FUNCTION_BLOCK FB_Robot
VAR_INPUT
	
	inint_NoOfJobs			: INT; 					(*	Number of Jobs / Numarul de module 	*)
	ins_CommIn				: Type_CommIn_Robot; 	(*	Communication Input for Robot / Modulele de comunicare pentru robot *)
	inint_OptNextJob		:INT;
	inm_Reset				:BOOL;
	
	inCom_0					:BOOL;	
	inCom_1					:BOOL;
	inCom_2					:BOOL;	
	inCom_3					:BOOL;	
	inCom_4					:BOOL;	
	inCom_5					:BOOL;	
	inCom_6					:BOOL;	
	inCom_7					:BOOL;	
	
	inCom_Re_0				:BYTE;
	inCom_Re_1				:BYTE;
	inCom_Re_2				:BYTE;
	inCom_Re_3				:BYTE;
	inCom_Re_4				:BYTE;
	inCom_Re_5				:BYTE;
	inCom_Re_6				:BYTE;
	inCom_Re_7				:BYTE;
	
	in_Opt					:Type_CommIn_Optimization;

END_VAR

VAR_OUTPUT

	outs_Order				: ENUM_OrderState;		(*	State of the order 0-Working / 1-Done / Starea actuala a piesei ridicate 0-in aer / 1-terminata *)
	outs_CommOut			: Type_CommOut_Robot;	(*	Communication output from robot / Comunicarea de la robot catre celelalte module *)
	m_Busy					: BOOL;					(*	Control variable that signals all the modules that robot is busy / o variabila de control ce semnalizeaza tuturor celorlalte module ca robotul este ocupat *)
	outs_Reset				: Type_CommOut_Reset;
	
	outs_Job				:ENUM_Order;
	outint_LastPosition		:INT;
	outdword_StartTime		:Type_Opt_Timers;
	outreal_AverageCycleTime:Type_Opt_CycleTime;
	out_Availabilty			:Type_OptIn_Availability;
	
	outCom_0				:BOOL 	:= m_CallRobotToModule[0];
	outCom_1				:BOOL	:= m_GoDownPick;
	outCom_2				:BOOL	:= m_CallRobotToModule[2];
	outCom_3				:BOOL	:= m_CallRobotToModule[3];
	outCom_4				:BOOL	:= m_CallRobotToModule[4];
	outCom_5				:BOOL	:= m_CallRobotToModule[5];
	outCom_6				:BOOL	:= m_CallRobotToModule[6];
	outCom_7				:BOOL	:= m_GoDownPlace;
	
	
	outCOm_Re_0				:BYTE;
	outCom_Re_1				:BYTE;
	outCom_Re_2				:BYTE;
	outCom_Re_3				:BYTE;
	outCom_Re_4				:BYTE	:=BOOL_TO_BYTE(m_CallRobotToModule[1]);
	outCom_Re_5				:BYTE;
	outCom_Re_6				:BYTE;
	outCom_Re_7				:BYTE;
	
	
END_VAR		

VAR
	Position		: ARRAY [0..11] OF BOOL; (*	Tine minte numarul modulului in dreptul caruia se afla robotul.In acelasi timp, 
											daca un index este egal cu 1, inseamna ca la modulul respectiv se va lucra,
											Se va face Pick sau Place*) 		
	int_Index				: INT;						(*	Index for memorizing the positions*)
	int_IndexForward		: INT;
	int_NextOrder			: ENUM_Order;				(*	*)
	int_PreviousOrder		: ENUM_Order;
	int_LastPosition		: INT;
	int_OptValue			: INT;
	MovementTimes			: ARRAY [0..50] OF TYPE_MovementTime;
	MovementTimesForward	: ARRAY [0..50] OF TYPE_MovementTime;
	m_BaseFinished			: BOOL :=TRUE;
	m_Picked				: BOOL;						(*	Daca robotul a executat miscarea de ridicare a piesei Down->Catch->Up, m_Picked devine true*)
	m_Placed				: BOOL;
	m_GoNextModule			: BOOL;						(*	Variabila de control pentru robot (in val3 citesc valoarea acestei variabile pentru a stii daca incep deplasarea sau nu)*)
	
	m_CallRobotToModule	:ARRAY[0..11] OF BOOL;		(*	Un array de bool prin care chem robotul la modulul la care am nevoie de el *)
	m_Condition			:BOOL;
	
	m_OptOn				:BOOL;
	
	T_Conveyor			:TON;
	T_Test1				:TON;
	T_Test2				:TON;
	T_Test3				:TON;
	T_Drilling1			:TON;
	T_Drilling			:TON;
	
	TC_StartTime		:DWORD;
	T1_StartTime		:DWORD;
	T2_StartTime		:DWORD;
	T3_StartTime		:DWORD;
	TD_StartTime		:DWORD;
	TD1_StartTime		:DWORD;
	
	T01_HelpTimer		:TON;
	T02_MoveTimer		:TON;
	T02_MoveTimer1		:TON;
	
	m_GoDownPick	:BOOL;	(*	Variabila ce transmite robotului ca poate face miscarea de pick*)
	m_GoDownPlace	:BOOL;	(*	Variabila ce transmite robotului ca poate face miscarea de place*)
	
	RetVal				: enum_RetVal;
	
	SFCInit 			:BOOL;
	(*-- Add IN/OUT for Robot Ethercat Communication	*)
	
	(* IN	*)	
	In_0_Byte_0_Bit_0	AT %I* 		:BOOL;
	In_0_Byte_0_Bit_1	AT %I* 		:BOOL;
	In_0_Byte_0_Bit_2	AT %I* 		:BOOL;
	In_0_Byte_0_Bit_3	AT %I* 		:BOOL;
	In_0_Byte_0_Bit_4	AT %I* 		:BOOL;
	In_0_Byte_0_Bit_5	AT %I* 		:BOOL;
	In_0_Byte_0_Bit_6	AT %I* 		:BOOL;
	In_0_Byte_0_Bit_7	AT %I* 		:BOOL;
	
	(* IN REAL*)
	
	inRe_0_Byte_0			AT %I*		:BYTE;
	inRe_0_Byte_1			AT %I*		:BYTE;
	inRe_0_Byte_2			AT %I*		:BYTE;
	inRe_0_Byte_3			AT %I*		:BYTE;
	inRe_0_Byte_4			AT %I*		:BYTE;
	inRe_0_Byte_5			AT %I*		:BYTE;
	inRe_0_Byte_6			AT %I*		:BYTE;
	inRe_0_Byte_7			AT %I*		:BYTE;


	(*	OUT	*)
	Out_0_Byte_0_Bit_0	AT %Q* 		:BOOL;
	Out_0_Byte_0_Bit_1	AT %Q* 		:BOOL;
	Out_0_Byte_0_Bit_2	AT %Q* 		:BOOL;
	Out_0_Byte_0_Bit_3	AT %Q* 		:BOOL;
	Out_0_Byte_0_Bit_4	AT %Q* 		:BOOL;
	Out_0_Byte_0_Bit_5	AT %Q* 		:BOOL;
	Out_0_Byte_0_Bit_6	AT %Q* 		:BOOL;
	Out_0_Byte_0_Bit_7	AT %Q* 		:BOOL;
	
	(* OUT REAL*)
	
	outRe_0_Byte_0			AT %Q*		:BYTE;
	outRe_0_Byte_1			AT %Q*		:BYTE;
	outRe_0_Byte_2			AT %Q*		:BYTE;
	outRe_0_Byte_3			AT %Q*		:BYTE;
	outRe_0_Byte_4			AT %Q*		:BYTE;
	outRe_0_Byte_5			AT %Q*		:BYTE;
	outRe_0_Byte_6			AT %Q*		:BYTE;
	outRe_0_Byte_7			AT %Q*		:BYTE;

	(*--											  --*)
	
	Inst_MovementTime			:FB_RobotMovementTime();
	Inst_MovementTimeBack		:FB_RobotMovementTime();
	
	Inst_Count5PiecesDone		:FB_CountCycleTime();
	real_PiecesTime				:REAL;
	int_PartsDone				:INT;	

END_VAR

A98_SetOutputs();
A99_Communication();

IF NOT inm_Reset 
	THEN
	m_Condition:=FALSE;
	Inst_MovementTime();
	Inst_MovementTimeBack();
	A02_AutomaticMode();
	
ELSIF inm_Reset 
	THEN
	
	IF NOT m_Condition
		THEN
		SFCReset:=TRUE;
		A02_AutomaticMode();		
	END_IF
	
	m_Condition:=TRUE;
	A03_S2_Reset();

END_IF

ACTION A02_AutomaticMode:
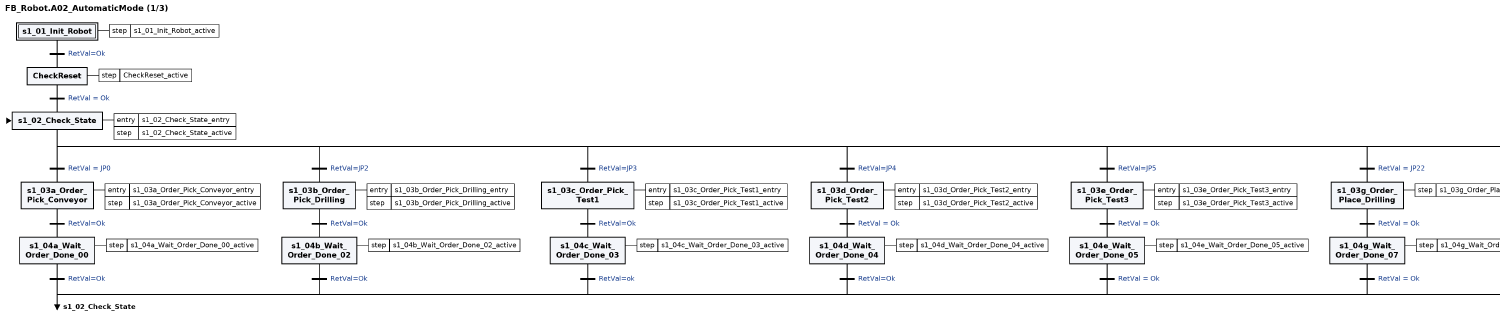
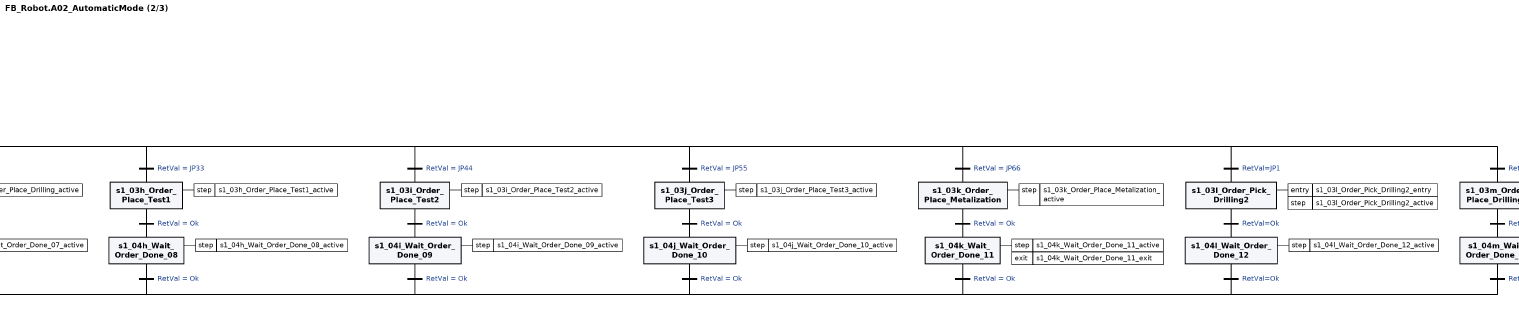
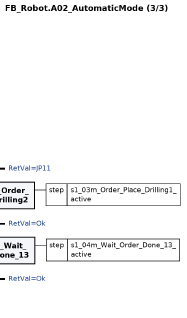
INITIAL_STEP s1_01_Init_Robot:
    s1_01_Init_Robot_active(N);  // step action
END_STEP
TRANSITION FROM s1_01_Init_Robot TO CheckReset
    := RetVal=Ok;
END_TRANSITION
STEP CheckReset:
    CheckReset_active(N);  // step action
END_STEP
TRANSITION FROM CheckReset TO s1_02_Check_State
    := RetVal = Ok;
END_TRANSITION
STEP s1_02_Check_State:
    s1_02_Check_State_entry(P1);  // entry action
    s1_02_Check_State_active(N);  // step action
END_STEP
TRANSITION FROM s1_02_Check_State TO s1_03a_Order_Pick_Conveyor
    := RetVal = JP0;
END_TRANSITION
STEP s1_03a_Order_Pick_Conveyor:
    s1_03a_Order_Pick_Conveyor_entry(P1);  // entry action
    s1_03a_Order_Pick_Conveyor_active(N);  // step action
END_STEP
TRANSITION FROM s1_03a_Order_Pick_Conveyor TO s1_04a_Wait_Order_Done_00
    := RetVal=Ok;
END_TRANSITION
STEP s1_04a_Wait_Order_Done_00:
    s1_04a_Wait_Order_Done_00_active(N);  // step action
END_STEP
TRANSITION FROM s1_04a_Wait_Order_Done_00 TO s1_02_Check_State
    := RetVal=Ok;
END_TRANSITION
TRANSITION FROM s1_02_Check_State TO s1_03b_Order_Pick_Drilling
    := RetVal=JP2;
END_TRANSITION
STEP s1_03b_Order_Pick_Drilling:
    s1_03b_Order_Pick_Drilling_entry(P1);  // entry action
    s1_03b_Order_Pick_Drilling_active(N);  // step action
END_STEP
TRANSITION FROM s1_03b_Order_Pick_Drilling TO s1_04b_Wait_Order_Done_02
    := RetVal=Ok;
END_TRANSITION
STEP s1_04b_Wait_Order_Done_02:
    s1_04b_Wait_Order_Done_02_active(N);  // step action
END_STEP
TRANSITION FROM s1_04b_Wait_Order_Done_02 TO s1_02_Check_State
    := RetVal=Ok;
END_TRANSITION
TRANSITION FROM s1_02_Check_State TO s1_03c_Order_Pick_Test1
    := RetVal=JP3;
END_TRANSITION
STEP s1_03c_Order_Pick_Test1:
    s1_03c_Order_Pick_Test1_entry(P1);  // entry action
    s1_03c_Order_Pick_Test1_active(N);  // step action
END_STEP
TRANSITION FROM s1_03c_Order_Pick_Test1 TO s1_04c_Wait_Order_Done_03
    := RetVal=Ok;
END_TRANSITION
STEP s1_04c_Wait_Order_Done_03:
    s1_04c_Wait_Order_Done_03_active(N);  // step action
END_STEP
TRANSITION FROM s1_04c_Wait_Order_Done_03 TO s1_02_Check_State
    := RetVal=ok;
END_TRANSITION
TRANSITION FROM s1_02_Check_State TO s1_03d_Order_Pick_Test2
    := RetVal=JP4;
END_TRANSITION
STEP s1_03d_Order_Pick_Test2:
    s1_03d_Order_Pick_Test2_entry(P1);  // entry action
    s1_03d_Order_Pick_Test2_active(N);  // step action
END_STEP
TRANSITION FROM s1_03d_Order_Pick_Test2 TO s1_04d_Wait_Order_Done_04
    := RetVal = Ok;
END_TRANSITION
STEP s1_04d_Wait_Order_Done_04:
    s1_04d_Wait_Order_Done_04_active(N);  // step action
END_STEP
TRANSITION FROM s1_04d_Wait_Order_Done_04 TO s1_02_Check_State
    := RetVal=Ok;
END_TRANSITION
TRANSITION FROM s1_02_Check_State TO s1_03e_Order_Pick_Test3
    := RetVal=JP5;
END_TRANSITION
STEP s1_03e_Order_Pick_Test3:
    s1_03e_Order_Pick_Test3_entry(P1);  // entry action
    s1_03e_Order_Pick_Test3_active(N);  // step action
END_STEP
TRANSITION FROM s1_03e_Order_Pick_Test3 TO s1_04e_Wait_Order_Done_05
    := RetVal = Ok;
END_TRANSITION
STEP s1_04e_Wait_Order_Done_05:
    s1_04e_Wait_Order_Done_05_active(N);  // step action
END_STEP
TRANSITION FROM s1_04e_Wait_Order_Done_05 TO s1_02_Check_State
    := RetVal = Ok;
END_TRANSITION
TRANSITION FROM s1_02_Check_State TO s1_03g_Order_Place_Drilling
    := RetVal = JP22;
END_TRANSITION
STEP s1_03g_Order_Place_Drilling:
    s1_03g_Order_Place_Drilling_active(N);  // step action
END_STEP
TRANSITION FROM s1_03g_Order_Place_Drilling TO s1_04g_Wait_Order_Done_07
    := RetVal = Ok;
END_TRANSITION
STEP s1_04g_Wait_Order_Done_07:
    s1_04g_Wait_Order_Done_07_active(N);  // step action
END_STEP
TRANSITION FROM s1_04g_Wait_Order_Done_07 TO s1_02_Check_State
    := RetVal = Ok;
END_TRANSITION
TRANSITION FROM s1_02_Check_State TO s1_03h_Order_Place_Test1
    := RetVal = JP33;
END_TRANSITION
STEP s1_03h_Order_Place_Test1:
    s1_03h_Order_Place_Test1_active(N);  // step action
END_STEP
TRANSITION FROM s1_03h_Order_Place_Test1 TO s1_04h_Wait_Order_Done_08
    := RetVal = Ok;
END_TRANSITION
STEP s1_04h_Wait_Order_Done_08:
    s1_04h_Wait_Order_Done_08_active(N);  // step action
END_STEP
TRANSITION FROM s1_04h_Wait_Order_Done_08 TO s1_02_Check_State
    := RetVal = Ok;
END_TRANSITION
TRANSITION FROM s1_02_Check_State TO s1_03i_Order_Place_Test2
    := RetVal = JP44;
END_TRANSITION
STEP s1_03i_Order_Place_Test2:
    s1_03i_Order_Place_Test2_active(N);  // step action
END_STEP
TRANSITION FROM s1_03i_Order_Place_Test2 TO s1_04i_Wait_Order_Done_09
    := RetVal = Ok;
END_TRANSITION
STEP s1_04i_Wait_Order_Done_09:
    s1_04i_Wait_Order_Done_09_active(N);  // step action
END_STEP
TRANSITION FROM s1_04i_Wait_Order_Done_09 TO s1_02_Check_State
    := RetVal = Ok;
END_TRANSITION
TRANSITION FROM s1_02_Check_State TO s1_03j_Order_Place_Test3
    := RetVal = JP55;
END_TRANSITION
STEP s1_03j_Order_Place_Test3:
    s1_03j_Order_Place_Test3_active(N);  // step action
END_STEP
TRANSITION FROM s1_03j_Order_Place_Test3 TO s1_04j_Wait_Order_Done_10
    := RetVal = Ok;
END_TRANSITION
STEP s1_04j_Wait_Order_Done_10:
    s1_04j_Wait_Order_Done_10_active(N);  // step action
END_STEP
TRANSITION FROM s1_04j_Wait_Order_Done_10 TO s1_02_Check_State
    := RetVal = Ok;
END_TRANSITION
TRANSITION FROM s1_02_Check_State TO s1_03k_Order_Place_Metalization
    := RetVal = JP66;
END_TRANSITION
STEP s1_03k_Order_Place_Metalization:
    s1_03k_Order_Place_Metalization_active(N);  // step action
END_STEP
TRANSITION FROM s1_03k_Order_Place_Metalization TO s1_04k_Wait_Order_Done_11
    := RetVal = Ok;
END_TRANSITION
STEP s1_04k_Wait_Order_Done_11:
    s1_04k_Wait_Order_Done_11_active(N);  // step action
    s1_04k_Wait_Order_Done_11_exit(P0);  // exit action
END_STEP
TRANSITION FROM s1_04k_Wait_Order_Done_11 TO s1_02_Check_State
    := RetVal = Ok;
END_TRANSITION
TRANSITION FROM s1_02_Check_State TO s1_03l_Order_Pick_Drilling2
    := RetVal=JP1;
END_TRANSITION
STEP s1_03l_Order_Pick_Drilling2:
    s1_03l_Order_Pick_Drilling2_entry(P1);  // entry action
    s1_03l_Order_Pick_Drilling2_active(N);  // step action
END_STEP
TRANSITION FROM s1_03l_Order_Pick_Drilling2 TO s1_04l_Wait_Order_Done_12
    := RetVal=Ok;
END_TRANSITION
STEP s1_04l_Wait_Order_Done_12:
    s1_04l_Wait_Order_Done_12_active(N);  // step action
END_STEP
TRANSITION FROM s1_04l_Wait_Order_Done_12 TO s1_02_Check_State
    := RetVal=Ok;
END_TRANSITION
TRANSITION FROM s1_02_Check_State TO s1_03m_Order_Place_Drilling2
    := RetVal=JP11;
END_TRANSITION
STEP s1_03m_Order_Place_Drilling2:
    s1_03m_Order_Place_Drilling1_active(N);  // step action
END_STEP
TRANSITION FROM s1_03m_Order_Place_Drilling2 TO s1_04m_Wait_Order_Done_13
    := RetVal=Ok;
END_TRANSITION
STEP s1_04m_Wait_Order_Done_13:
    s1_04m_Wait_Order_Done_13_active(N);  // step action
END_STEP
TRANSITION FROM s1_04m_Wait_Order_Done_13 TO s1_02_Check_State
    := RetVal=Ok;
END_TRANSITION
// branch label Branch0_A01_AutomaticMode
END_ACTION

ACTION A03_S2_Reset:
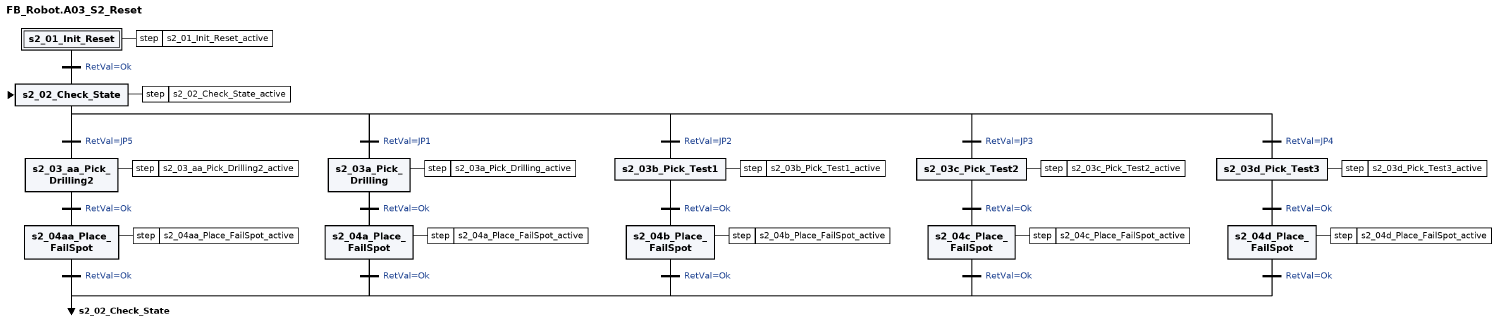
INITIAL_STEP s2_01_Init_Reset:
    s2_01_Init_Reset_active(N);  // step action
END_STEP
TRANSITION FROM s2_01_Init_Reset TO s2_02_Check_State
    := RetVal=Ok;
END_TRANSITION
STEP s2_02_Check_State:
    s2_02_Check_State_active(N);  // step action
END_STEP
TRANSITION FROM s2_02_Check_State TO s2_03_aa_Pick_Drilling2
    := RetVal=JP5;
END_TRANSITION
STEP s2_03_aa_Pick_Drilling2:
    s2_03_aa_Pick_Drilling2_active(N);  // step action
END_STEP
TRANSITION FROM s2_03_aa_Pick_Drilling2 TO s2_04aa_Place_FailSpot
    := RetVal=Ok;
END_TRANSITION
STEP s2_04aa_Place_FailSpot:
    s2_04aa_Place_FailSpot_active(N);  // step action
END_STEP
TRANSITION FROM s2_04aa_Place_FailSpot TO s2_02_Check_State
    := RetVal=Ok;
END_TRANSITION
TRANSITION FROM s2_02_Check_State TO s2_03a_Pick_Drilling
    := RetVal=JP1;
END_TRANSITION
STEP s2_03a_Pick_Drilling:
    s2_03a_Pick_Drilling_active(N);  // step action
END_STEP
TRANSITION FROM s2_03a_Pick_Drilling TO s2_04a_Place_FailSpot
    := RetVal=Ok;
END_TRANSITION
STEP s2_04a_Place_FailSpot:
    s2_04a_Place_FailSpot_active(N);  // step action
END_STEP
TRANSITION FROM s2_04a_Place_FailSpot TO s2_02_Check_State
    := RetVal=Ok;
END_TRANSITION
TRANSITION FROM s2_02_Check_State TO s2_03b_Pick_Test1
    := RetVal=JP2;
END_TRANSITION
STEP s2_03b_Pick_Test1:
    s2_03b_Pick_Test1_active(N);  // step action
END_STEP
TRANSITION FROM s2_03b_Pick_Test1 TO s2_04b_Place_FailSpot
    := RetVal=Ok;
END_TRANSITION
STEP s2_04b_Place_FailSpot:
    s2_04b_Place_FailSpot_active(N);  // step action
END_STEP
TRANSITION FROM s2_04b_Place_FailSpot TO s2_02_Check_State
    := RetVal=Ok;
END_TRANSITION
TRANSITION FROM s2_02_Check_State TO s2_03c_Pick_Test2
    := RetVal=JP3;
END_TRANSITION
STEP s2_03c_Pick_Test2:
    s2_03c_Pick_Test2_active(N);  // step action
END_STEP
TRANSITION FROM s2_03c_Pick_Test2 TO s2_04c_Place_FailSpot
    := RetVal=Ok;
END_TRANSITION
STEP s2_04c_Place_FailSpot:
    s2_04c_Place_FailSpot_active(N);  // step action
END_STEP
TRANSITION FROM s2_04c_Place_FailSpot TO s2_02_Check_State
    := RetVal=Ok;
END_TRANSITION
TRANSITION FROM s2_02_Check_State TO s2_03d_Pick_Test3
    := RetVal=JP4;
END_TRANSITION
STEP s2_03d_Pick_Test3:
    s2_03d_Pick_Test3_active(N);  // step action
END_STEP
TRANSITION FROM s2_03d_Pick_Test3 TO s2_04d_Place_FailSpot
    := RetVal=Ok;
END_TRANSITION
STEP s2_04d_Place_FailSpot:
    s2_04d_Place_FailSpot_active(N);  // step action
END_STEP
TRANSITION FROM s2_04d_Place_FailSpot TO s2_02_Check_State
    := RetVal=Ok;
END_TRANSITION
// branch label Branch0_A03_S2_Reset
END_ACTION

ACTION A98_SetOutputs:
outCom_0	:= inCom_0;
outCom_1 	:= inCom_1;
outCom_2 	:= inCom_2;
outCom_3 	:= inCom_3;
outCom_4 	:= inCom_4;
outCom_5	:= inCom_5;
outCom_6 	:= inCom_6;
outCom_7 	:= inCom_7;


outCom_Re_0	:= inCom_Re_0;
outCom_Re_1	:= inCom_Re_1;
outCom_Re_2	:= inCom_Re_2;
outCom_Re_3	:= inCom_Re_3;
outCom_Re_4	:= inCom_Re_4;
outCom_Re_5	:= inCom_Re_5;
outCom_Re_6	:= inCom_Re_6;
outCom_Re_7	:= inCom_Re_7;
END_ACTION

ACTION A99_Communication:

(*inputs*)

Position[0] 	:= In_0_Byte_0_Bit_0;
m_Picked 		:= In_0_Byte_0_Bit_1;
Position[2]  	:= In_0_Byte_0_Bit_2;
Position[3]  	:= In_0_Byte_0_Bit_3;
Position[4]  	:= In_0_Byte_0_Bit_4;
Position[5]  	:= In_0_Byte_0_Bit_5;
Position[6]  	:= In_0_Byte_0_Bit_6;
m_Placed 		:= In_0_Byte_0_Bit_7;


inCom_Re_0		:= inRe_0_Byte_0;
inCom_Re_1		:= inRe_0_Byte_1;
inCom_Re_2		:= inRe_0_Byte_2;
inCom_Re_3		:= inRe_0_Byte_3;
Position[1]		:= BYTE_TO_BOOL(inRe_0_Byte_4);
m_OptOn			:= BYTE_TO_BOOL(inRe_0_Byte_5);
inCom_Re_6		:= inRe_0_Byte_6;
inCom_Re_7		:= inRe_0_Byte_7;

(*outputs*)

Out_0_Byte_0_Bit_0 	:= m_CallRobotToModule[0];
Out_0_Byte_0_Bit_1 	:= m_GoDownPick;
Out_0_Byte_0_Bit_2 	:= m_CallRobotToModule[2];
Out_0_Byte_0_Bit_3 	:= m_CallRobotToModule[3];
Out_0_Byte_0_Bit_4	:= m_CallRobotToModule[4];
Out_0_Byte_0_Bit_5 	:= m_CallRobotToModule[5];
Out_0_Byte_0_Bit_6 	:= m_CallRobotToModule[6];
Out_0_Byte_0_Bit_7 	:= m_GoDownPlace;

outRe_0_Byte_0		:= outCom_Re_0;
outRe_0_Byte_1		:= outCom_Re_1;
outRe_0_Byte_2		:= outCom_Re_2;
outRe_0_Byte_3		:= outCom_Re_3;
outRe_0_Byte_4		:= BOOL_TO_BYTE(m_CallRobotToModule[1]);
outRe_0_Byte_5		:= INT_TO_BYTE(int_OptValue);
outRe_0_Byte_6		:= outCom_Re_6;
outRe_0_Byte_7		:= outCom_Re_7;

outdword_StartTime.T_Conveyor	:=TC_StartTime;
outdword_StartTime.T_Drilling_1	:=TD1_StartTime;
outdword_StartTime.T_Drilling	:=TD_StartTime;
outdword_StartTime.T_Test_1		:=T1_StartTime;
outdword_StartTime.T_Test_2		:=T2_StartTime;
outdword_StartTime.T_Test_3		:=T3_StartTime;

outreal_AverageCycleTime.re_Conveyor	:=in_Opt.s_Conveyor.out_AverageCycleTime;
outreal_AverageCycleTime.re_Drilling_1	:=in_Opt.s_Drilling_1.out_AverageCycleTime;
outreal_AverageCycleTime.re_Drilling	:=in_Opt.s_Drilling_2.out_AverageCycleTime;
outreal_AverageCycleTime.re_Test_1		:=in_Opt.s_Test_1.out_AverageCycleTime;
outreal_AverageCycleTime.re_Test_2		:=in_Opt.s_Test_2.out_AverageCycleTime;
outreal_AverageCycleTime.re_Test_3		:=in_Opt.s_Test_3.out_AverageCycleTime;

out_Availabilty.s_Drilling_1.m_Available	:= ins_CommIn.s_Drilling.m_Empty;
out_Availabilty.s_Drilling_2.m_Available	:= ins_CommIn.s_Drilling1.m_Empty;
out_Availabilty.s_Test_1.m_Available		:= ins_CommIn.s_Test_1.m_Empty;
out_Availabilty.s_Test_2.m_Available		:= ins_CommIn.s_Test_2.m_Empty;
out_Availabilty.s_Test_3.m_Available		:= ins_CommIn.s_Test_3.m_Empty;
out_Availabilty.s_Metalization.m_Available	:= ins_CommIn.s_Metalization.m_Empty;

outint_LastPosition	:=int_LastPosition;
outs_Job			:=int_NextOrder;
END_ACTION

ACTION CheckReset_active:
RetVal	:=Running;

IF 	NOT inm_Reset
	THEN
	RetVal	:=Ok;
END_IF
END_ACTION

ACTION s1_01_Init_Robot_active:
IF m_BaseFinished
	THEN	
		Inst_Count5PiecesDone(inm_TimeActive:=TRUE);
		
		outs_Order:=ENUM_OrderState.Done;
		
		outs_CommOut.s_Conveyor.m_OutOfArea		:=TRUE;
		outs_CommOut.s_Drilling.m_OutOfArea		:=TRUE;	
		outs_CommOut.s_Drilling1.m_OutOfArea	:=TRUE;	
		outs_CommOut.s_Test_1.m_OutOfArea		:=TRUE;
		outs_CommOut.s_Test_2.m_OutOfArea		:=TRUE;
		outs_CommOut.s_Test_3.m_OutOfArea		:=TRUE;
		outs_CommOut.s_Metalization.m_OutOfArea	:=TRUE;
		
		outs_Reset.outm_Reset_Drilling	:=FALSE;
		outs_Reset.outm_Reset_Drilling2	:=FALSE;
		outs_Reset.outm_Reset_Test1		:=FALSE;
		outs_Reset.outm_Reset_Test2		:=FALSE;
		outs_Reset.outm_Reset_Test3		:=FALSE;

		T1_StartTime:=T2_StartTime:=T3_StartTime:=	TIME_TO_DWORD(T#1D) + 20000;
		TD1_StartTime:=TD_StartTime:=TC_StartTime:= TIME_TO_DWORD(T#1D);
		
		RetVal:=Ok;
		
		
			
END_IF
END_ACTION

ACTION s1_02_Check_State_active:

(* 	----PICK TEST1,TEST2,TEST3----	*)

	IF (	T1_StartTime<T2_StartTime
		AND 	T1_StartTime<T3_StartTime)
		AND 	ins_CommIn.s_Test_1.m_Ready
		AND 	ins_CommIn.s_Metalization.m_Empty
		AND NOT m_Picked
		AND (
				int_NextOrder = ENUM_Order.NoOrder
		OR		int_NextOrder = ENUM_Order.Pick_Test_1)
		THEN
			int_NextOrder:=ENUM_Order.Pick_Test_1;
			RetVal := JP3;	
			
	
	ELSIF 	(	T2_StartTime<T1_StartTime
		AND 	T2_StartTime<T3_StartTime)
		AND 	ins_CommIn.s_Test_2.m_Ready
		AND 	ins_CommIn.s_Metalization.m_Empty
		AND NOT m_Picked
		AND (
				int_NextOrder = ENUM_Order.NoOrder
		OR		int_NextOrder = ENUM_Order.Pick_Test_2)
		THEN
			int_NextOrder:=ENUM_Order.Pick_Test_2;
			RetVal := JP4;	
			
	ELSIF 	(	T3_StartTime<T1_StartTime
		AND 	T3_StartTime<T2_StartTime)
		AND 	ins_CommIn.s_Test_3.m_Ready
		AND 	ins_CommIn.s_Metalization.m_Empty	
		AND NOT m_Picked
		AND (
				int_NextOrder = ENUM_Order.NoOrder
		OR		int_NextOrder = ENUM_Order.Pick_Test_3)
		THEN
			int_NextOrder:=ENUM_Order.Pick_Test_3;
			RetVal := JP5;	
	
	
			
	(* 	----PICK DRILLING1,DRILLING2----	*)	
	ELSIF 	TD_StartTime<TD1_StartTime
		AND (	ins_CommIn.s_Drilling.m_Ready
		AND (	ins_CommIn.s_Test_1.m_Empty
			OR 	ins_CommIn.s_Test_2.m_Empty
			OR 	ins_CommIn.s_Test_3.m_Empty
			)
		AND NOT m_Picked
		AND
			( 	int_NextOrder = ENUM_Order.NoOrder 
		OR		int_NextOrder = ENUM_Order.Pick_Drilling)
			)
		THEN
			int_NextOrder:=ENUM_Order.Pick_Drilling;
			RetVal := JP2;
				
	ELSIF 		TD1_StartTime<TD_StartTime
		AND (	ins_CommIn.s_Drilling1.m_Ready
		AND (	ins_CommIn.s_Test_1.m_Empty
			OR 	ins_CommIn.s_Test_2.m_Empty
			OR 	ins_CommIn.s_Test_3.m_Empty
			)
		AND NOT m_Picked
		AND
			( 	int_NextOrder = ENUM_Order.NoOrder 
		OR		int_NextOrder = ENUM_Order.Pick_Drilling1)
			)
		THEN
			int_NextOrder:=ENUM_Order.Pick_Drilling1;
			RetVal := JP1;
			
	(* 	----PICK CONVEYOR----	*)			
	ELSIF		(ins_CommIn.s_Conveyor.m_Ready (* verific daca modulul actual are piesa gata	*)
		AND 	(ins_CommIn.s_Drilling.m_Empty (* verific daca urmatorul modul e gol	(altfel nu fac pick de aici)	*)
		OR		 ins_CommIn.s_Drilling1.m_Empty)
		AND NOT m_Picked	
		AND
			(	int_NextOrder=ENUM_Order.NoOrder 
		OR 		int_NextOrder=ENUM_Order.Pick_Conveyor)
			)
		THEN
			int_NextOrder:=ENUM_Order.Pick_Conveyor;
			RetVal:=JP0;
				
	(*	PLACE	*)
	
	ELSIF 	ins_CommIn.s_Drilling1.m_Empty
		AND m_Picked	
		AND outs_Order = ENUM_OrderState.Done
		AND m_GoNextModule
		AND
		(	int_NextOrder = ENUM_Order.NoOrder 	
		OR	int_NextOrder = ENUM_Order.Place_Drilling2)	
		
		THEN
			RetVal := JP11;
			
	ELSIF 	ins_CommIn.s_Drilling.m_Empty
		AND m_Picked	
		AND outs_Order = ENUM_OrderState.Done
		AND m_GoNextModule
		AND
		(	int_NextOrder = ENUM_Order.NoOrder 	
		OR	int_NextOrder = ENUM_Order.Place_Drilling)	
		
		THEN
			RetVal := JP22;
	
	ELSIF 	ins_CommIn.s_Test_1.m_Empty
		AND m_Picked
		AND NOT m_Busy	
		AND outs_Order = ENUM_OrderState.Done
		AND m_GoNextModule
		AND
		(	int_NextOrder = ENUM_Order.NoOrder 	
		OR	int_NextOrder = ENUM_Order.Place_Test_1)	
		
		THEN
			RetVal := JP33;
		
	ELSIF 	ins_CommIn.s_Test_2.m_Empty
		AND m_Picked
		AND NOT m_Busy	
		AND outs_Order = ENUM_OrderState.Done
		AND m_GoNextModule
		AND
		(	int_NextOrder = ENUM_Order.NoOrder 	
		OR	int_NextOrder = ENUM_Order.Place_Test_2)	
		
		THEN
			RetVal := JP44;
			
	ELSIF 	ins_CommIn.s_Test_3.m_Empty
		AND m_Picked
		AND NOT m_Busy	
		AND outs_Order = ENUM_OrderState.Done
		AND m_GoNextModule
		AND
		(	int_NextOrder = ENUM_Order.NoOrder 	
		OR	int_NextOrder = ENUM_Order.Place_Test_3)	
		
		THEN
			RetVal := JP55;
			
		
	ELSIF 	ins_CommIn.s_Metalization.m_Empty 
		AND m_Picked
		AND outs_Order = ENUM_OrderState.Done
		AND m_GoNextModule
		AND 
		(	int_NextOrder = ENUM_Order.NoOrder
		OR	int_NextOrder = ENUM_Order.Place_Metalization)
		
		THEN
			RetVal := JP66;
	
	END_IF
END_ACTION

ACTION s1_02_Check_State_entry:
RetVal:= Running;

IF m_OptOn AND int_NextOrder=ENUM_Order.NoOrder
	THEN
	int_OptValue:= inint_OptNextJob;
	
	CASE int_OptValue OF
		0:	int_NextOrder := ENUM_Order.Pick_Conveyor;
		1:	int_NextOrder := ENUM_Order.Pick_Drilling1;
		2:	int_NextOrder := ENUM_Order.Pick_Drilling;
		3:	int_NextOrder := ENUM_Order.Pick_Test_1;
		4:	int_NextOrder := ENUM_Order.Pick_Test_2;
		5:	int_NextOrder := ENUM_Order.Pick_Test_3;
	END_CASE
	
END_IF
			
IF int_NextOrder=ENUM_Order.Pick_Conveyor
		AND ins_CommIn.s_Conveyor.m_Ready 
		THEN
			RetVal:=JP0;
			
	ELSIF int_NextOrder=ENUM_Order.Pick_Drilling
		AND ins_CommIn.s_Drilling.m_Ready 
		THEN
			RetVal:=JP2;
			
	ELSIF int_NextOrder=ENUM_Order.Pick_Drilling1
		AND ins_CommIn.s_Drilling1.m_Ready 
		THEN
			RetVal:=JP1;
			
	ELSIF int_NextOrder=ENUM_Order.Pick_Test_1
		AND ins_CommIn.s_Test_1.m_Ready 
		THEN
			RetVal:=JP3;
	ELSIF int_NextOrder=ENUM_Order.Pick_Test_2
		AND ins_CommIn.s_Test_2.m_Ready 
		THEN
			RetVal:=JP4;
	ELSIF int_NextOrder=ENUM_Order.Pick_Test_3
		AND ins_CommIn.s_Test_3.m_Ready 
		THEN
			RetVal:=JP5;
	END_IF
END_ACTION

ACTION s1_03a_Order_Pick_Conveyor_active:
RetVal:=Running;
outs_CommOut.s_Metalization.m_OutOfArea:=TRUE;
(* semnal pentru urmatorul modul ca robotul lucreaza *)
m_CallRobotToModule[0] := TRUE; (*	Chem robotul la conveyor.Aceasta variabila trebuie sa o citesc in programul robotului*)

outs_Order:=ENUM_OrderState.Working; 
outs_CommOut.s_Conveyor.m_Work:=TRUE;(*	Semnalez conveyorul ca robotul urmeaza sa lucreze in jurul lui	*)
T_Conveyor(IN:=FALSE);
IF Position[0] = 1
	THEN
		Inst_MovementTimeBack(inm_Couting:=FALSE, inint_SecondStation:=0);
		MovementTimes[int_Index].FirstStation := Inst_MovementTimeBack.outs_MovementTime.FirstStation;
		MovementTimes[int_Index].SecondStation := Inst_MovementTimeBack.outs_MovementTime.SecondStation;
		MovementTimes[int_Index].MovementTime := Inst_MovementTimeBack.outs_MovementTime.MovementTime;
		outs_CommOut.s_Conveyor.m_OutOfArea:=FALSE;	
		// Trebuie o variabila care sa dea startul miscarii de pick sau de place. m_GoDown
				(*	In acest punct, robotul a luat piesa si este sus ,m_Picked este conctrolat din staubli*)		
END_IF

IF ins_CommIn.s_Conveyor.m_Ready
		THEN		
	m_GoDownPick:=TRUE;	
	IF m_Picked
	THEN
		m_CallRobotToModule[0]	:=	FALSE;
		outs_CommOut.s_Conveyor.m_Work:=FALSE;	
		m_GoDownPick:= FALSE; 	//aici se face FALSE pentru a nu ramane mereu activa.
		TC_StartTime:=TIME_TO_DWORD(T_Conveyor.StartTime);
		int_Index:=int_Index + 1;		
		RetVal :=Ok;						
		END_IF
END_IF
 (*-----------IAR M_PICKED SE VA FACE TRUE IN STAUBLI---------------------------------------*)

// La final... Next order trebuie sa fie de place pe urmatorul modul int_NextOrder:=ENUM_Order.Place_Drilling;




(*	Miscarea	


	Order = Pick	=> 	Move From Initial Position To Asked Position 	--Gloval_Vars.Order[] 
						Move Down To Take Part							--m_MoveDown 
						Move Up With Part								--m_MoveUp	=>m_Picked
					
	Order = Place	=>	Move From Last Position To Asked Position		-Global_Vars.Order[]
						Move Down To Leave Part							--m_MoveDown
						Move Up Empty									--m_MoveUp	=>m_Placed	
						
	
	SAU
	
	
	Order = Pick 	=> Logica facuta in Staubli include MoveToTarget, MoveDown, MoveUp
	*)
END_ACTION

ACTION s1_03a_Order_Pick_Conveyor_entry:
Inst_MovementTimeBack(inm_Couting:=TRUE, inint_FirstStation:=int_LastPosition);
T_Conveyor(IN:=TRUE);
END_ACTION

ACTION s1_03b_Order_Pick_Drilling_active:
RetVal:=Running;
outs_CommOut.s_Metalization.m_OutOfArea:=TRUE;
int_PreviousOrder:= ENUM_Order.Pick_Drilling;
m_CallRobotToModule[2] := TRUE; 
outs_Order:=ENUM_OrderState.Working; 
outs_CommOut.s_Drilling.m_Work:=TRUE;

IF Position[2] = 1
	THEN	
		Inst_MovementTimeBack(inm_Couting:=FALSE, inint_SecondStation:=2);
		MovementTimes[int_Index].FirstStation := Inst_MovementTimeBack.outs_MovementTime.FirstStation;
		MovementTimes[int_Index].SecondStation := Inst_MovementTimeBack.outs_MovementTime.SecondStation;
		MovementTimes[int_Index].MovementTime := Inst_MovementTimeBack.outs_MovementTime.MovementTime;
		outs_CommOut.s_Drilling.m_OutOfArea:=FALSE;
				
		m_GoDownPick	:=TRUE;		
END_IF

		
IF m_Picked (*	m_Picked este controlata din staubli	*)
		THEN
			m_CallRobotToModule[2]	:=	FALSE;
			outs_CommOut.s_Drilling.m_PartDropped:=FALSE;
			outs_CommOut.s_Drilling.m_Work:=FALSE;
			m_GoDownPick:=FALSE;		
			int_Index:=int_Index + 1;	
			RetVal := Ok;
END_IF
END_ACTION

ACTION s1_03b_Order_Pick_Drilling_entry:
Inst_MovementTimeBack(inm_Couting:=TRUE, inint_FirstStation:=int_LastPosition);
END_ACTION

ACTION s1_03c_Order_Pick_Test1_active:
RetVal:=Running;
outs_CommOut.s_Metalization.m_OutOfArea:=TRUE;
int_PreviousOrder := ENUM_Order.Pick_Test_1;
m_CallRobotToModule[3] := TRUE; 
outs_Order:=ENUM_OrderState.Working; (* inseamna ca piesa e in aer *)
outs_CommOut.s_Test_1.m_Work:=TRUE;
 
IF Position[3] = 1
	THEN
		Inst_MovementTimeBack(inm_Couting:=FALSE, inint_SecondStation:=3);
		MovementTimes[int_Index].FirstStation := Inst_MovementTimeBack.outs_MovementTime.FirstStation;
		MovementTimes[int_Index].SecondStation := Inst_MovementTimeBack.outs_MovementTime.SecondStation;
		MovementTimes[int_Index].MovementTime := Inst_MovementTimeBack.outs_MovementTime.MovementTime;
		outs_CommOut.s_Test_1.m_OutOfArea:=FALSE;
	m_GoDownPick	:=TRUE;	
END_IF
	
			
IF m_Picked (*	m_Picked este controlata din staubli	*)
		THEN
			m_CallRobotToModule[3]	:=	FALSE;
			outs_CommOut.s_Test_1.m_PartDropped:=FALSE;
			outs_CommOut.s_Test_1.m_Work:=FALSE;
			m_GoDownPick:=FALSE;
			int_Index:=int_Index + 1;			
			RetVal := Ok;
END_IF

 
// La final... Next order trebuie sa fie de place pe urmatorul modul int_NextOrder:=ENUM_Order.Place_Drilling;




(*	Miscarea	


	Order = Pick	=> 	Move From Initial Position To Asked Position 	--Gloval_Vars.Order[] 
						Move Down To Take Part							--m_MoveDown 
						Move Up With Part								--m_MoveUp	=>m_Picked
					
	Order = Place	=>	Move From Last Position To Asked Position		-Global_Vars.Order[]
						Move Down To Leave Part							--m_MoveDown
						Move Up Empty									--m_MoveUp	=>m_Placed	
						
	
	SAU
	
	
	Order = Pick 	=> Logica facuta in Staubli include MoveToTarget, MoveDown, MoveUp
	*)
END_ACTION

ACTION s1_03c_Order_Pick_Test1_entry:
Inst_MovementTimeBack(inm_Couting:=TRUE, inint_FirstStation:=int_LastPosition);
END_ACTION

ACTION s1_03d_Order_Pick_Test2_active:
RetVal:=Running;
outs_CommOut.s_Metalization.m_OutOfArea:=TRUE;
(* semnal pentru urmatorul modul ca robotul lucreaza *)
int_PreviousOrder := ENUM_Order.Pick_Test_2;
m_CallRobotToModule[4] := TRUE; 
outs_Order:=ENUM_OrderState.Working; (* inseamna ca piesa e in aer *)
outs_CommOut.s_Test_2.m_Work:=TRUE;

IF Position[4] = 1
	THEN
		Inst_MovementTimeBack(inm_Couting:=FALSE, inint_SecondStation:=4);
		MovementTimes[int_Index].FirstStation := Inst_MovementTimeBack.outs_MovementTime.FirstStation;
		MovementTimes[int_Index].SecondStation := Inst_MovementTimeBack.outs_MovementTime.SecondStation;
		MovementTimes[int_Index].MovementTime := Inst_MovementTimeBack.outs_MovementTime.MovementTime;
		
		outs_CommOut.s_Test_2.m_OutOfArea:=FALSE;
		
	
		m_GoDownPick	:=TRUE;
	

END_IF


	IF m_Picked (*	m_Picked este controlata din staubli	*)
		THEN
			m_CallRobotToModule[4]	:=	FALSE;
			outs_CommOut.s_Test_2.m_PartDropped:=FALSE;
			outs_CommOut.s_Test_2.m_Work:=FALSE;
			m_GoDownPick:=FALSE;	
			int_Index:=int_Index + 1;		
			RetVal := Ok;
	END_IF


 
// La final... Next order trebuie sa fie de place pe urmatorul modul int_NextOrder:=ENUM_Order.Place_Drilling;




(*	Miscarea	


	Order = Pick	=> 	Move From Initial Position To Asked Position 	--Gloval_Vars.Order[] 
						Move Down To Take Part							--m_MoveDown 
						Move Up With Part								--m_MoveUp	=>m_Picked
					
	Order = Place	=>	Move From Last Position To Asked Position		-Global_Vars.Order[]
						Move Down To Leave Part							--m_MoveDown
						Move Up Empty									--m_MoveUp	=>m_Placed	
						
	
	SAU
	
	
	Order = Pick 	=> Logica facuta in Staubli include MoveToTarget, MoveDown, MoveUp
	*)
END_ACTION

ACTION s1_03d_Order_Pick_Test2_entry:
Inst_MovementTimeBack(inm_Couting:=TRUE, inint_FirstStation:=int_LastPosition);
END_ACTION

ACTION s1_03e_Order_Pick_Test3_active:
RetVal:=Running;
outs_CommOut.s_Metalization.m_OutOfArea:=TRUE;
(* semnal pentru urmatorul modul ca robotul lucreaza *)
int_PreviousOrder := ENUM_Order.Pick_Test_3;
m_CallRobotToModule[5] := TRUE; 
outs_Order:=ENUM_OrderState.Working; (* inseamna ca piesa e in aer *)
outs_CommOut.s_Test_3.m_Work:=TRUE;


IF Position[5] = 1
	THEN
		Inst_MovementTimeBack(inm_Couting:=FALSE, inint_SecondStation:=5);
		MovementTimes[int_Index].FirstStation := Inst_MovementTimeBack.outs_MovementTime.FirstStation;
		MovementTimes[int_Index].SecondStation := Inst_MovementTimeBack.outs_MovementTime.SecondStation;
		MovementTimes[int_Index].MovementTime := Inst_MovementTimeBack.outs_MovementTime.MovementTime;
		
		outs_CommOut.s_Test_3.m_OutOfArea:=FALSE;
			m_GoDownPick:=TRUE;

END_IF

	IF m_Picked (*	m_Picked este controlata din staubli	*)
	THEN
		m_CallRobotToModule[5]	:=	FALSE;
		outs_CommOut.s_Test_3.m_PartDropped:=FALSE;
		outs_CommOut.s_Test_3.m_Work:=FALSE;
		m_GoDownPick:=FALSE;
		int_Index:=int_Index + 1;			
		RetVal := Ok;
	END_IF


 
// La final... Next order trebuie sa fie de place pe urmatorul modul int_NextOrder:=ENUM_Order.Place_Drilling;
END_ACTION

ACTION s1_03e_Order_Pick_Test3_entry:
Inst_MovementTimeBack(inm_Couting:=TRUE, inint_FirstStation:=int_LastPosition);
END_ACTION

ACTION s1_03f_Order_Pick_Metalization_active:

END_ACTION

ACTION s1_03g_Order_Place_Drilling_active:
RetVal:=Running;
m_CallRobotToModule[2] :=	TRUE; (*	Adica robotul e chemat la drilling	*)
outs_CommOut.s_Conveyor.m_OutOfArea:=TRUE;
T_Drilling(IN:=FALSE);
outs_Order:=ENUM_OrderState.Working;

outs_CommOut.s_Drilling.m_Work:=TRUE;

IF m_GoNextModule 		(*	Daca e adevarat, robotul are permisiunea de a merge la modulul urmator*)		
	THEN
		
	IF Position[2] = 1
		THEN 	
			Inst_MovementTime(inm_Couting:=FALSE, inint_SecondStation:=2);
			MovementTimesForward[int_IndexForward].FirstStation := Inst_MovementTime.outs_MovementTime.FirstStation;
			MovementTimesForward[int_IndexForward].SecondStation := Inst_MovementTime.outs_MovementTime.SecondStation;
			MovementTimesForward[int_IndexForward].MovementTime := Inst_MovementTime.outs_MovementTime.MovementTime;

			m_GoDownPlace:=TRUE;
			outs_CommOut.s_Drilling.m_OutOfArea:=FALSE;
	END_IF

	IF m_Placed
		THEN	
			int_IndexForward:=int_IndexForward + 1;
			m_CallRobotToModule[2]	:=	FALSE;
			T_Drilling(IN:=TRUE);		
			TD_StartTime:=TIME_TO_DWORD(T_Drilling.StartTime);
			outs_CommOut.s_Drilling.m_Work:=FALSE;
			m_GoDownPlace:=FALSE;
			RetVal := Ok;
	END_IF
END_IF

(*	La final next order trebuie sa fie no order !!!*)
END_ACTION

ACTION s1_03h_Order_Place_Test1_active:
RetVal:=Running;
m_CallRobotToModule[3] :=	TRUE; (*	Adica robotul e chemat la drilling	*)
IF int_PreviousOrder = ENUM_Order.Pick_Drilling
	THEN
	outs_CommOut.s_Drilling.m_OutOfArea:=TRUE;
ELSIF int_PreviousOrder = ENUM_Order.Pick_Drilling1
	THEN
	outs_CommOut.s_Drilling1.m_OutOfArea:=TRUE;
END_IF
T_Test1(IN:=FALSE);
outs_Order:=ENUM_OrderState.Working;

outs_CommOut.s_Test_1.m_Work:=TRUE;

IF m_GoNextModule 		(*	Daca e adevarat, robotul are permisiunea de a merge la modulul urmator*)		
	THEN
			
	IF Position[3] = 1
		THEN 	
			Inst_MovementTime(inm_Couting:=FALSE, inint_SecondStation:=3);
			MovementTimesForward[int_IndexForward].FirstStation := Inst_MovementTime.outs_MovementTime.FirstStation;
			MovementTimesForward[int_IndexForward].SecondStation := Inst_MovementTime.outs_MovementTime.SecondStation;
			MovementTimesForward[int_IndexForward].MovementTime := Inst_MovementTime.outs_MovementTime.MovementTime;

			m_GoDownPlace:=TRUE;
			outs_CommOut.s_Test_1.m_OutOfArea:=FALSE;
	END_IF

	IF m_Placed
		THEN
			m_CallRobotToModule[3]	:=	FALSE;
			int_IndexForward:=int_IndexForward + 1;
			T_Test1(IN:=TRUE);		
			T1_StartTime:=TIME_TO_DWORD(T_Test1.StartTime);
			outs_CommOut.s_Test_1.m_Work:=FALSE;
			m_GoDownPlace:=FALSE;
			RetVal := Ok;
	END_IF
END_IF

(*	La final next order trebuie sa fie no order !!!*)
END_ACTION

ACTION s1_03i_Order_Place_Test2_active:
RetVal:=Running;
m_CallRobotToModule[4] :=	TRUE; (*	Adica robotul e chemat la drilling	*)
IF int_PreviousOrder = ENUM_Order.Pick_Drilling
	THEN
	outs_CommOut.s_Drilling.m_OutOfArea:=TRUE;
ELSIF int_PreviousOrder = ENUM_Order.Pick_Drilling1
	THEN
	outs_CommOut.s_Drilling1.m_OutOfArea:=TRUE;
END_IF
T_Test2(IN:=FALSE);
outs_Order:=ENUM_OrderState.Working;

outs_CommOut.s_Test_2.m_Work:=TRUE;

IF m_GoNextModule 		(*	Daca e adevarat, robotul are permisiunea de a merge la modulul urmator*)		
	THEN
	
	IF Position[4] = 1
		THEN 	
			Inst_MovementTime(inm_Couting:=FALSE, inint_SecondStation:=4);
			MovementTimesForward[int_IndexForward].FirstStation := Inst_MovementTime.outs_MovementTime.FirstStation;
			MovementTimesForward[int_IndexForward].SecondStation := Inst_MovementTime.outs_MovementTime.SecondStation;
			MovementTimesForward[int_IndexForward].MovementTime := Inst_MovementTime.outs_MovementTime.MovementTime;

			m_GoDownPlace:=TRUE;
			outs_CommOut.s_Test_2.m_OutOfArea:=FALSE;
	END_IF

	IF m_Placed
		THEN
			int_IndexForward:=int_IndexForward + 1;
			m_CallRobotToModule[4]	:=	FALSE;
			T_Test2(IN:=TRUE);		
			T2_StartTime:=TIME_TO_DWORD(T_Test2.StartTime);
			outs_CommOut.s_Test_2.m_Work:=FALSE;
			m_GoDownPlace:=FALSE;
			RetVal := Ok;
	END_IF
END_IF

(*	La final next order trebuie sa fie no order !!!*)
END_ACTION

ACTION s1_03j_Order_Place_Test3_active:
RetVal:=Running;
m_CallRobotToModule[5] :=	TRUE; (*	Adica robotul e chemat la drilling	*)
IF int_PreviousOrder = ENUM_Order.Pick_Drilling
	THEN
	outs_CommOut.s_Drilling.m_OutOfArea:=TRUE;
ELSIF int_PreviousOrder = ENUM_Order.Pick_Drilling1
	THEN
	outs_CommOut.s_Drilling1.m_OutOfArea:=TRUE;
END_IF
T_Test3(IN:=FALSE);
outs_Order:=ENUM_OrderState.Working;

outs_CommOut.s_Test_3.m_Work:=TRUE;

(*
	--Comunicarea dintre robot si plc prin biti.			
*)

IF m_GoNextModule 		(*	Daca e adevarat, robotul are permisiunea de a merge la modulul urmator*)		
	THEN
	(*	
		--Miscarea catre pozitia 02.
		Position[2] := 1;
	*)
			
	IF Position[5] = 1
		THEN 	
			Inst_MovementTime(inm_Couting:=FALSE, inint_SecondStation:=5);
			MovementTimesForward[int_IndexForward].FirstStation := Inst_MovementTime.outs_MovementTime.FirstStation;
			MovementTimesForward[int_IndexForward].SecondStation := Inst_MovementTime.outs_MovementTime.SecondStation;
			MovementTimesForward[int_IndexForward].MovementTime := Inst_MovementTime.outs_MovementTime.MovementTime;

			m_GoDownPlace:=TRUE;
			outs_CommOut.s_Test_3.m_OutOfArea:=FALSE;
	END_IF

	IF m_Placed
		THEN
			int_IndexForward:=int_IndexForward + 1;
			m_CallRobotToModule[5]	:=	FALSE;
			T_Test3(IN:=TRUE);		
			T3_StartTime:=TIME_TO_DWORD(T_Test3.StartTime);
			outs_CommOut.s_Test_3.m_Work:=FALSE;
			m_GoDownPlace:=FALSE;
			RetVal := Ok;
	END_IF
END_IF

(*	La final next order trebuie sa fie no order !!!*)
END_ACTION

ACTION s1_03k_Order_Place_Metalization_active:
RetVal:=Running;
m_CallRobotToModule[6] 	:=	TRUE; (*	Adica robotul e chemat la drilling	*)

outs_Order:=ENUM_OrderState.Working;

IF 		int_PreviousOrder = ENUM_Order.Pick_Test_1
	THEN
	outs_CommOut.s_Test_1.m_OutOfArea:=TRUE;
ELSIF	int_PreviousOrder = ENUM_Order.Pick_Test_2
	THEN
	outs_CommOut.s_Test_2.m_OutOfArea:=TRUE;
ELSIF	int_PreviousOrder = ENUM_Order.Pick_Test_3
	THEN
	outs_CommOut.s_Test_3.m_OutOfArea:=TRUE;
END_IF
	
outs_CommOut.s_Metalization.m_Work:=TRUE;
(*
	--Comunicarea dintre robot si plc prin biti.			
*)

IF m_GoNextModule 		(*	Daca e adevarat, robotul are permisiunea de a merge la modulul urmator*)		
	THEN
	(*	
		--Miscarea catre pozitia 02.
		Position[2] := 1;
	*)
			
	IF Position[6] = 1
		THEN 	
			Inst_MovementTime(inm_Couting:=FALSE, inint_SecondStation:=6);
				MovementTimesForward[int_IndexForward].FirstStation := Inst_MovementTime.outs_MovementTime.FirstStation;
			MovementTimesForward[int_IndexForward].SecondStation := Inst_MovementTime.outs_MovementTime.SecondStation;
			MovementTimesForward[int_IndexForward].MovementTime := Inst_MovementTime.outs_MovementTime.MovementTime;

			m_GoDownPlace:=TRUE;
			outs_CommOut.s_Metalization.m_OutOfArea:=FALSE;
	END_IF

	IF m_Placed
		THEN
			int_IndexForward:=int_IndexForward + 1;
			m_CallRobotToModule[6]	:=	FALSE;
			outs_CommOut.s_Metalization.m_Work:=FALSE;
			m_GoDownPlace:=FALSE;
			RetVal := Ok;
	END_IF
END_IF

(*	La final next order trebuie sa fie no order !!!*)
END_ACTION

ACTION s1_03l_Order_Pick_Drilling2_active:
RetVal:=Running;
outs_CommOut.s_Metalization.m_OutOfArea:=TRUE;
int_PreviousOrder:= ENUM_Order.Pick_Drilling1;
m_CallRobotToModule[1] := TRUE; 
outs_Order:=ENUM_OrderState.Working; 
outs_CommOut.s_Drilling1.m_Work:=TRUE;

IF Position[1] = 1
	THEN	
		Inst_MovementTimeBack(inm_Couting:=FALSE, inint_SecondStation:=1);
		MovementTimes[int_Index].FirstStation := Inst_MovementTimeBack.outs_MovementTime.FirstStation;
		MovementTimes[int_Index].SecondStation := Inst_MovementTimeBack.outs_MovementTime.SecondStation;
		MovementTimes[int_Index].MovementTime := Inst_MovementTimeBack.outs_MovementTime.MovementTime;
		outs_CommOut.s_Drilling1.m_OutOfArea:=FALSE;
		m_GoDownPick:=TRUE;
END_IF

IF m_Picked (*	m_Picked este controlata din staubli	*)
	THEN
		m_CallRobotToModule[1]	:=	FALSE;
		outs_CommOut.s_Drilling1.m_PartDropped:=FALSE;
		outs_CommOut.s_Drilling1.m_Work:=FALSE;
		m_GoDownPick:=FALSE;		
		int_Index:=int_Index + 1;	
		RetVal := Ok;
END_IF
END_ACTION

ACTION s1_03l_Order_Pick_Drilling2_entry:
Inst_MovementTimeBack(inm_Couting:=TRUE, inint_FirstStation:=int_LastPosition);
END_ACTION

ACTION s1_03m_Order_Place_Drilling1_active:
RetVal:=Running;
m_CallRobotToModule[1] :=	TRUE; (*	Adica robotul e chemat la drilling	*)
outs_CommOut.s_Conveyor.m_OutOfArea:=TRUE;
T_Drilling1(IN:=FALSE);
outs_Order:=ENUM_OrderState.Working;

outs_CommOut.s_Drilling1.m_Work:=TRUE;

IF m_GoNextModule 		(*	Daca e adevarat, robotul are permisiunea de a merge la modulul urmator*)		
	THEN
		
	IF Position[1] = 1
		THEN 	
			Inst_MovementTime(inm_Couting:=FALSE, inint_SecondStation:=1);
			MovementTimesForward[int_IndexForward].FirstStation := Inst_MovementTime.outs_MovementTime.FirstStation;
			MovementTimesForward[int_IndexForward].SecondStation := Inst_MovementTime.outs_MovementTime.SecondStation;
			MovementTimesForward[int_IndexForward].MovementTime := Inst_MovementTime.outs_MovementTime.MovementTime;

			m_GoDownPlace:=TRUE;
			outs_CommOut.s_Drilling1.m_OutOfArea:=FALSE;
	END_IF

	IF m_Placed
		THEN	
			int_IndexForward:=int_IndexForward + 1;
			m_CallRobotToModule[1]	:=	FALSE;
			T_Drilling1(IN:=TRUE);		
			TD1_StartTime:=TIME_TO_DWORD(T_Drilling1.StartTime);
			outs_CommOut.s_Drilling1.m_Work:=FALSE;
			m_GoDownPlace:=FALSE;
			RetVal := Ok;
	END_IF
END_IF

(*	La final next order trebuie sa fie no order !!!*)
END_ACTION

ACTION s1_04a_Wait_Order_Done_00_active:
RetVal := Running;
IF ins_CommIn.s_Drilling.m_Empty
	THEN
	int_NextOrder	:=ENUM_Order.Place_Drilling;
ELSIF ins_CommIn.s_Drilling1.m_Empty
	THEN
	int_NextOrder	:=ENUM_Order.Place_Drilling2;	
END_IF

Inst_MovementTime(inm_Couting:=TRUE, inint_FirstStation:=0);

m_GoNextModule := TRUE;		

IF ins_CommIn.s_Conveyor.m_Ready = FALSE (*	Conveyorul nu poate fi ready din nou, decat daca robotul a plecat de acolo *)
	THEN
	RetVal:=Ok;
END_IF


outs_Order		:=ENUM_OrderState.Done; 			(* 	Inseamna ca piesa este ridicata (deci orderul a fost indeplinit)	*)
END_ACTION

ACTION s1_04b_Wait_Order_Done_02_active:
RetVal := Running;

IF ins_CommIn.s_Test_1.m_Empty
	THEN
		int_NextOrder:=ENUM_Order.Place_Test_1;
ELSIF ins_CommIn.s_Test_2.m_Empty
	THEN
		int_NextOrder:=ENUM_Order.Place_Test_2;
ELSIF ins_CommIn.s_Test_3.m_Empty
	THEN
		int_NextOrder:=ENUM_Order.Place_Test_3;
END_IF

Inst_MovementTime(inm_Couting:=TRUE, inint_FirstStation:=2);
m_GoNextModule:=TRUE;

IF ins_CommIn.s_Drilling.m_Ready = FALSE
	THEN
	RetVal:=Ok;
END_IF

outs_Order		:=ENUM_OrderState.Done; 			(* 	Inseamna ca piesa este ridicata (deci orderul a fost indeplinit)	*)
END_ACTION

ACTION s1_04c_Wait_Order_Done_03_active:
RetVal := Running;

int_NextOrder:=ENUM_Order.Place_Metalization;
Inst_MovementTime(inm_Couting:=TRUE, inint_FirstStation:=3);
m_GoNextModule:=TRUE;

IF ins_CommIn.s_Test_1.m_Ready = FALSE	
	THEN
	RetVal:=Ok;
END_IF

outs_Order		:=ENUM_OrderState.Done; 			(* 	Inseamna ca piesa este ridicata (deci orderul a fost indeplinit)	*)
END_ACTION

ACTION s1_04d_Wait_Order_Done_04_active:
RetVal := Running;

int_NextOrder:=ENUM_Order.Place_Metalization;
Inst_MovementTime(inm_Couting:=TRUE, inint_FirstStation:=4);
m_GoNextModule:=TRUE;

IF ins_CommIn.s_Test_2.m_Ready = FALSE
	THEN	
	RetVal:=Ok;
END_IF

outs_Order		:=ENUM_OrderState.Done; 			(* 	Inseamna ca piesa este ridicata (deci orderul a fost indeplinit)	*)
END_ACTION

ACTION s1_04e_Wait_Order_Done_05_active:
RetVal := Running;

int_NextOrder:=ENUM_Order.Place_Metalization;
Inst_MovementTime(inm_Couting:=TRUE, inint_FirstStation:=5);

m_GoNextModule:=TRUE;
(*	In acest punct piesa este in aer trebuie dusa la modul --- pe alta ramura(alt step)*)

(*	Comunicat la robot sa mearga la urmatorul modul (Drilling) 
	
	
	
	In momentul in care piesa a fost luata de pe modul, modulul trebuie sa lucreze din nou, 
	deci iesirea lui trebuie sa fie m_ready = FALSE;
	
	Inseamna ca piesa a fost intradevar luata, iar alta poate intra in prelucrare(asta trebuie facuta in modul)
	Position[0] := 0; 
	
*)


(*	Mai trebuie un pas intermediar in care robotul elibereaza zona de lucru a conveyorului
	inainte de a intra pe stepul de place.*)
 


IF ins_CommIn.s_Test_3.m_Ready = FALSE
	THEN
	RetVal:=Ok;
END_IF

outs_Order		:=ENUM_OrderState.Done; 			(* 	Inseamna ca piesa este ridicata (deci orderul a fost indeplinit)	*)
END_ACTION

ACTION s1_04f_Wait_Order_Done_06_active:

END_ACTION

ACTION s1_04g_Wait_Order_Done_07_active:
RetVal:=Running;

outs_Order:=ENUM_OrderState.Done;

int_NextOrder:=ENUM_Order.NoOrder;
int_LastPosition := 2;
m_GoNextModule:=FALSE;
	
IF ins_CommIn.s_Drilling.m_Empty = FALSE
	THEN
	outs_CommOut.s_Drilling.m_OutOfArea:=TRUE;
	outs_CommOut.s_Drilling.m_PartDropped:=TRUE;
	RetVal:=Ok;
END_IF
END_ACTION

ACTION s1_04h_Wait_Order_Done_08_active:
RetVal:=Running;

outs_Order:=ENUM_OrderState.Done;

int_NextOrder:=ENUM_Order.NoOrder;
int_LastPosition := 3;
m_GoNextModule:=FALSE;
	
IF ins_CommIn.s_Test_1.m_Empty = FALSE
	THEN
	outs_CommOut.s_Test_1.m_OutOfArea:=TRUE;
	outs_CommOut.s_Test_1.m_PartDropped:=TRUE;
	RetVal:=Ok;
END_IF
END_ACTION

ACTION s1_04i_Wait_Order_Done_09_active:
RetVal:=Running;

outs_Order:=ENUM_OrderState.Done;

int_NextOrder:=ENUM_Order.NoOrder;
int_LastPosition := 4;
m_GoNextModule:=FALSE;
	
IF ins_CommIn.s_Test_2.m_Empty = FALSE
	THEN
	outs_CommOut.s_Test_2.m_OutOfArea:=TRUE;
	outs_CommOut.s_Test_2.m_PartDropped:=TRUE;
	RetVal:=Ok;
END_IF
END_ACTION

ACTION s1_04j_Wait_Order_Done_10_active:
RetVal:=Running;

outs_Order:=ENUM_OrderState.Done;

int_NextOrder:=ENUM_Order.NoOrder;
int_LastPosition := 5;
m_GoNextModule:=FALSE;
	
IF ins_CommIn.s_Test_3.m_Empty = FALSE
	THEN
	outs_CommOut.s_Test_3.m_OutOfArea:=TRUE;
	outs_CommOut.s_Test_3.m_PartDropped:=TRUE;

	RetVal:=Ok;
END_IF
END_ACTION

ACTION s1_04k_Wait_Order_Done_11_active:
RetVal:=Running;

outs_Order:=ENUM_OrderState.Done;

int_NextOrder:=ENUM_Order.NoOrder;
int_LastPosition := 6;
m_GoNextModule:=FALSE;

IF ins_CommIn.s_Metalization.m_Empty = FALSE
	THEN
	outs_CommOut.s_Metalization.m_OutOfArea:=TRUE;
	outs_CommOut.s_Metalization.m_PartDropped:=TRUE;
	int_PartsDone:=int_PartsDone+1;
	RetVal:=Ok;
END_IF
END_ACTION

ACTION s1_04k_Wait_Order_Done_11_exit:
outs_CommOut.s_Metalization.m_PartDropped:=FALSE;

IF int_PartsDone=5
	THEN
	Inst_Count5PiecesDone(inm_TimeActive:=FALSE);
	real_PiecesTime:=Inst_Count5PiecesDone.outr_CycleTime;
END_IF
END_ACTION

ACTION s1_04l_Wait_Order_Done_12_active:
RetVal := Running;

IF ins_CommIn.s_Test_1.m_Empty
	THEN
		int_NextOrder:=ENUM_Order.Place_Test_1;
ELSIF ins_CommIn.s_Test_2.m_Empty
	THEN
		int_NextOrder:=ENUM_Order.Place_Test_2;
ELSIF ins_CommIn.s_Test_3.m_Empty
	THEN
		int_NextOrder:=ENUM_Order.Place_Test_3;
END_IF

Inst_MovementTime(inm_Couting:=TRUE, inint_FirstStation:=1);
m_GoNextModule:=TRUE;

IF ins_CommIn.s_Drilling1.m_Ready = FALSE
	THEN
	RetVal:=Ok;
END_IF

outs_Order		:=ENUM_OrderState.Done; 			(* 	Inseamna ca piesa este ridicata (deci orderul a fost indeplinit)	*)
END_ACTION

ACTION s1_04m_Wait_Order_Done_13_active:
RetVal:=Running;

outs_Order:=ENUM_OrderState.Done;

int_NextOrder:=ENUM_Order.NoOrder;
int_LastPosition := 1;
m_GoNextModule:=FALSE;
	
IF ins_CommIn.s_Drilling1.m_Empty = FALSE
	THEN
	outs_CommOut.s_Drilling1.m_OutOfArea:=TRUE;
	outs_CommOut.s_Drilling1.m_PartDropped:=TRUE;
	RetVal:=Ok;
END_IF
END_ACTION

ACTION s2_01_Init_Reset_active:
RetVal:=Running;
SFCReset:=FALSE;

IF inm_Reset
	THEN	
	RetVal:=Ok;			
END_IF
END_ACTION

ACTION s2_02_Check_State_active:
RetVal:= Running;

IF 			ins_CommIn.s_Drilling.m_Ready (* verific daca modulul actual are piesa gata	*)
	AND NOT m_Picked	
	THEN
		RetVal:=JP1;
ELSIF		ins_CommIn.s_Drilling1.m_Ready
	AND NOT m_Picked
	THEN
		RetVal:=JP5;		
ELSIF		ins_CommIn.s_Test_1.m_Ready
	AND NOT m_Picked
	THEN
		RetVal:=JP2;
		
ELSIF		ins_CommIn.s_Test_2.m_Ready
	AND NOT m_Picked
	THEN
		RetVal:=JP3;		
		
ELSIF		ins_CommIn.s_Test_3.m_Ready
	AND NOT m_Picked
	THEN
		RetVal:=JP4;		
END_IF
END_ACTION

ACTION s2_03_aa_Pick_Drilling2_active:
RetVal:=Running;

m_CallRobotToModule[1] := TRUE; 

IF Position[1] = 1
	THEN	
		m_GoDownPick:=TRUE;
END_IF

IF m_Picked 
	THEN
		m_GoNextModule:=TRUE;
		m_CallRobotToModule[1]	:=	FALSE;
		m_GoDownPick:=FALSE;	
		outs_CommOut.s_Drilling1.m_PartDropped:=FALSE;
		outs_Reset.outm_Reset_Drilling2:=TRUE;	
		RetVal := Ok;
		
END_IF
END_ACTION

ACTION s2_03a_Pick_Drilling_active:
RetVal:=Running;

m_CallRobotToModule[2] := TRUE; 

IF Position[2] = 1
	THEN	
		m_GoDownPick:=TRUE;
END_IF

IF m_Picked 
	THEN
		m_GoNextModule:=TRUE;
		m_CallRobotToModule[2]	:=	FALSE;
		m_GoDownPick:=FALSE;	
		outs_CommOut.s_Drilling.m_PartDropped:=FALSE;
		outs_Reset.outm_Reset_Drilling:=TRUE;	
		RetVal := Ok;
		
END_IF
END_ACTION

ACTION s2_03b_Pick_Test1_active:
RetVal:=Running;

m_CallRobotToModule[3] := TRUE; 

IF Position[3] = 1
	THEN	
		m_GoDownPick:=TRUE;
END_IF

IF m_Picked 
	THEN
		m_GoNextModule:=TRUE;
		m_CallRobotToModule[3]	:=	FALSE;
		m_GoDownPick:=FALSE;	
		outs_CommOut.s_Test_1.m_PartDropped:=FALSE;
		outs_Reset.outm_Reset_Test1:=TRUE;			
		RetVal := Ok;
END_IF
END_ACTION

ACTION s2_03c_Pick_Test2_active:
RetVal:=Running;

m_CallRobotToModule[4] := TRUE; 

IF Position[4] = 1
	THEN	
		m_GoDownPick:=TRUE;
END_IF

IF m_Picked 
	THEN
		m_GoNextModule:=TRUE;
		m_CallRobotToModule[4]	:=	FALSE;
		m_GoDownPick:=FALSE;	
		outs_CommOut.s_Test_2.m_PartDropped:=FALSE;
		outs_Reset.outm_Reset_Test2:=TRUE;			
		RetVal := Ok;
END_IF
END_ACTION

ACTION s2_03d_Pick_Test3_active:
RetVal:=Running;

m_CallRobotToModule[5] := TRUE; 

IF Position[5] = 1
	THEN	
		m_GoDownPick:=TRUE;
END_IF

IF m_Picked 
	THEN
		m_GoNextModule:=TRUE;
		m_CallRobotToModule[5]	:=	FALSE;
		m_GoDownPick:=FALSE;	
		outs_CommOut.s_Test_3.m_PartDropped:=FALSE;
		outs_Reset.outm_Reset_Test3:=TRUE;			
		RetVal := Ok;
END_IF
END_ACTION

ACTION s2_04a_Place_FailSpot_active:
RetVal:=Running;

IF m_GoNextModule 			
	THEN			
	IF m_Placed
		THEN
			outs_Reset.outm_Reset_Drilling:=FALSE;	
			m_GoDownPlace:=FALSE;
			RetVal := Ok;
	END_IF
END_IF
END_ACTION

ACTION s2_04aa_Place_FailSpot_active:
RetVal:=Running;

IF m_GoNextModule 			
	THEN			
	IF m_Placed
		THEN
			outs_Reset.outm_Reset_Drilling2:=FALSE;	
			m_GoDownPlace:=FALSE;
			RetVal := Ok;
	END_IF
END_IF
END_ACTION

ACTION s2_04b_Place_FailSpot_active:
RetVal:=Running;

IF m_GoNextModule 			
	THEN			
	IF m_Placed
		THEN
			outs_Reset.outm_Reset_Test1:=FALSE;	
			m_GoDownPlace:=FALSE;
			RetVal := Ok;
	END_IF
END_IF
END_ACTION

ACTION s2_04c_Place_FailSpot_active:
RetVal:=Running;

IF m_GoNextModule 			
	THEN			
	IF m_Placed
		THEN
			outs_Reset.outm_Reset_Test2:=FALSE;	
			m_GoDownPlace:=FALSE;
			RetVal := Ok;
	END_IF
END_IF
END_ACTION

ACTION s2_04d_Place_FailSpot_active:
RetVal:=Running;

IF m_GoNextModule 			
	THEN			
	IF m_Placed
		THEN
			outs_Reset.outm_Reset_Test3:=FALSE;	
			m_GoDownPlace:=FALSE;
			RetVal := Ok;
	END_IF
END_IF
END_ACTION

END_FUNCTION_BLOCK

(* stored: Version 1.1.0.1, ProductVersion 3.1.4024.3
   POU FB_Robot: Id {2fc510c2-b84d-4206-9321-9c30fadb25a0}, SpecialFunc None
   Folder S1: Id {4a2f7b83-552c-48f8-a37f-880fcfe71f35}
   Folder 0_Pick: Id {db82c1d3-3c2b-4adf-b760-c8b04c7769b7}
   Folder 1_Place: Id {f925fc57-65f7-415b-b9ab-1caefbe7d66f}
   Folder S2: Id {46a90108-7be4-4beb-89f3-bc79487dfd60}
   Action A02_AutomaticMode: Id {2ea1cfad-ee6a-4f99-a19c-ef8c3f06be67}
   Action A03_S2_Reset: Id {124c9f31-6843-4cb3-97b9-608c4b2ca1c2}
   Action A98_SetOutputs: Id {6089db03-f1fd-4101-91a1-3b94529e70bc}
   Action A99_Communication: Id {4debeec3-6eee-4c77-9ab9-3291919af488}
   Action CheckReset_active: Id {ca9099e5-c386-4557-97bc-1cce1d10788f}
   Action s1_01_Init_Robot_active: Id {3a5d87bf-fd85-4d14-a902-0f380c060d9f}
   Action s1_02_Check_State_active: Id {d32dbc1e-6ff3-4478-bb9c-377cd2e76afc}
   Action s1_02_Check_State_entry: Id {f175980b-7b3a-4195-b9ac-88c0dcf16688}
   Action s1_03a_Order_Pick_Conveyor_active: Id {26dba430-ac14-4200-87ba-c09c6b67e2f2}
   Action s1_03a_Order_Pick_Conveyor_entry: Id {7da34524-faec-430e-9c9a-4d49372ef360}
   Action s1_03b_Order_Pick_Drilling_active: Id {36eadd8e-0f11-4ae9-8452-93c130a8dce7}
   Action s1_03b_Order_Pick_Drilling_entry: Id {c891c612-94a2-4141-9ed2-bbe97aa19401}
   Action s1_03c_Order_Pick_Test1_active: Id {c1f38a72-7d28-4d73-873a-b8fd541ba2da}
   Action s1_03c_Order_Pick_Test1_entry: Id {3fc9cbc4-ba13-4ad0-a17f-c7f66f96a7c4}
   Action s1_03d_Order_Pick_Test2_active: Id {6b6340d1-2f2b-4c56-8a7e-968a145281bf}
   Action s1_03d_Order_Pick_Test2_entry: Id {0cf7a8c7-810f-4f72-895c-b25b6f045702}
   Action s1_03e_Order_Pick_Test3_active: Id {0f2e4902-5ad5-4c12-9f2b-eaa075803b2c}
   Action s1_03e_Order_Pick_Test3_entry: Id {04a66867-e927-4bef-9cdc-d626cb48d1f0}
   Action s1_03f_Order_Pick_Metalization_active: Id {2e503a11-994b-416b-a1c7-44a56760f20f}
   Action s1_03g_Order_Place_Drilling_active: Id {6a444b04-8276-415c-9d20-caa4660e0c08}
   Action s1_03h_Order_Place_Test1_active: Id {6d849f8e-d3e9-4ae9-b294-b5a6dc5bbc5c}
   Action s1_03i_Order_Place_Test2_active: Id {a25642fc-a41e-4573-8460-4d911f59f455}
   Action s1_03j_Order_Place_Test3_active: Id {5f5f5c7c-8c78-40ca-9af2-9096a7607112}
   Action s1_03k_Order_Place_Metalization_active: Id {2c9b9eb9-3e3f-4cf4-8979-0a59b6e1b36a}
   Action s1_03l_Order_Pick_Drilling2_active: Id {9601529b-2b39-4aa1-bba1-4020963c2043}
   Action s1_03l_Order_Pick_Drilling2_entry: Id {d7bd983f-cce4-4508-8d80-a0bf73ff40b8}
   Action s1_03m_Order_Place_Drilling1_active: Id {8c13b9d1-41ed-4623-bbc1-d0840bdbda63}
   Action s1_04a_Wait_Order_Done_00_active: Id {9eeb5666-1f6b-45fc-b836-202af841d160}
   Action s1_04b_Wait_Order_Done_02_active: Id {d97f2b20-5892-4f42-9d9e-2dffaba5c23f}
   Action s1_04c_Wait_Order_Done_03_active: Id {f91ae87e-01b1-4c8c-8fc7-8a002643a97f}
   Action s1_04d_Wait_Order_Done_04_active: Id {4aa9c810-8d46-438a-b47d-4faf0155e110}
   Action s1_04e_Wait_Order_Done_05_active: Id {b0af9220-84b3-486e-909c-cdf3c27ce858}
   Action s1_04f_Wait_Order_Done_06_active: Id {3c4b8f92-1c10-42d9-98a0-9061e3cfe39e}
   Action s1_04g_Wait_Order_Done_07_active: Id {f5bd433e-5aae-4006-85de-4dc8c73e7f47}
   Action s1_04h_Wait_Order_Done_08_active: Id {9aeff2fb-ecfc-4d67-a0b1-2804bedd322d}
   Action s1_04i_Wait_Order_Done_09_active: Id {776f3afc-835a-46af-8ee6-0ab57d267d1e}
   Action s1_04j_Wait_Order_Done_10_active: Id {b0020a5e-a468-4f4e-9daf-21c041a82993}
   Action s1_04k_Wait_Order_Done_11_active: Id {723516dc-05f7-4df7-bf70-381f93189fb7}
   Action s1_04k_Wait_Order_Done_11_exit: Id {24dbdd42-cad8-4d8b-a479-0bdd954b5415}
   Action s1_04l_Wait_Order_Done_12_active: Id {cae149aa-f715-4d89-99b0-c8ddcacfebfe}
   Action s1_04m_Wait_Order_Done_13_active: Id {7361a221-edc9-461a-8682-7fab02617214}
   Action s2_01_Init_Reset_active: Id {6936803b-7d74-480e-aca4-cce8d2652632}
   Action s2_02_Check_State_active: Id {552316da-5e1b-4f8f-a727-4244a79a3a55}
   Action s2_03_aa_Pick_Drilling2_active: Id {c0d4d906-72e8-4d78-adf5-e5cbc74fe522}
   Action s2_03a_Pick_Drilling_active: Id {7777dad2-b76c-4905-bed3-0053b58a09d1}
   Action s2_03b_Pick_Test1_active: Id {4267dd6a-e9b4-412c-9b93-de26712f3e5e}
   Action s2_03c_Pick_Test2_active: Id {63145869-e6c2-45e7-b459-4a5fa2cb36bb}
   Action s2_03d_Pick_Test3_active: Id {74f9155b-1552-4451-bd0b-c7c6bf5a8c40}
   Action s2_04a_Place_FailSpot_active: Id {58f1a77a-892d-4db8-a743-8ff8331d86cf}
   Action s2_04aa_Place_FailSpot_active: Id {c45b93e7-ae3d-46c7-a358-1b58d0cf229e}
   Action s2_04b_Place_FailSpot_active: Id {f2910a45-553e-4b1a-8354-2d6bbd09dcf8}
   Action s2_04c_Place_FailSpot_active: Id {2ded11bb-66f3-46e4-bbc0-a494c49217c2}
   Action s2_04d_Place_FailSpot_active: Id {49c776fd-da9b-4078-80bc-f6ac144cf991} *)
